// TIA Portal V17 export
// export: Created 2024-06-16T17:47:19.2348542Z, ExportSetting WithDefaults, DisplayName Totally Integrated Automation Portal, DisplayVersion V17, DisplayName TIA Portal Openness, DisplayVersion V17, DisplayName TIA Portal Version Control Interface, DisplayVersion V17, DisplayName STEP 7 Professional, DisplayVersion V17, DisplayName STEP 7 Safety, DisplayVersion V17, DisplayName WinCC Professional, DisplayVersion V17
DATA_BLOCK "St0_In"   // DB5
{ S7_Optimized_Access := 'TRUE' }
VERSION : 0.1
// stored: AutoNumber false, DBAccessibleFromOPCUA true, DBAccessibleFromWebserver true, IsOnlyStoredInLoadMemory false, IsRetainMemResEnabled false, IsWriteProtectedInAS false, MemoryReserve 100
   VAR
      AU_1 : Bool;   // Arrêt d'urgence n°1
      AU_2 : Bool;   // Arrêt d'urgence n°2
      BP_Rearm : Bool;   // Réarmement machine
      Barillet_MP : Bool;   // Barillet Métaux Précieux ouvert (MP)
      PorteEntree_Fermee : Bool;   // Porte d'entrée : Fermée
      PorteSortie_Fermee : Bool;   // Porte de sortie : Fermée
      PorteVision_Fermee : Bool;   // Porte maintenance vision façade : Fermée
      PorteArriere_Fermee : Bool;   // Portes maitenance arrière machine : Fermée
   END_VAR
BEGIN
END_DATA_BLOCK
